FUNCTION_BLOCK ConveyorManualISub (* Conveyor Manual Interface subscribe *)
  (* Standard: 61499-2 *)
  (* Version 0.2, 2003-12-05, JHC, Rockwell Automation, Renamed from NEWCOMPFB. *)
  (* Version 0.1, 2002-01-08, JHC, Rockwell Automation, Added DLY FB as example. *)
  (* Version 0.0, 2000-05-27, JHC, Rockwell Automation *)
  (* Compiler header: package fb.rt.dasdA1.A2.Conveyor; *)
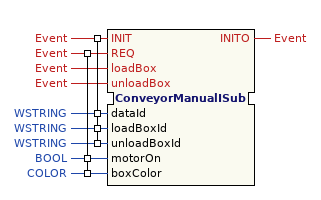
  EVENT_INPUT
    INIT WITH dataId, loadBoxId, unloadBoxId; (* Initialization Request *)
    REQ WITH motorOn, boxColor;
    loadBox;
    unloadBox;
  END_EVENT
  EVENT_OUTPUT
    INITO; (* Initialization Confirm *)
  END_EVENT
  VAR_INPUT
    dataId : WSTRING;
    loadBoxId : WSTRING;
    unloadBoxId : WSTRING;
    motorOn : BOOL;
    boxColor : COLOR;
  END_VAR
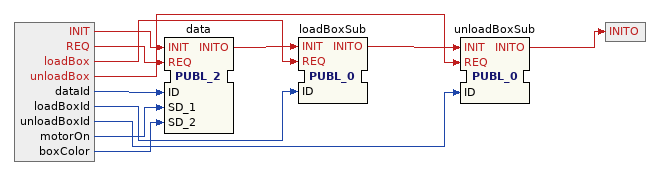
  FBS
    data : PUBL_2;
    loadBoxSub : PUBL_0;
    unloadBoxSub : PUBL_0;
  END_FBS
  EVENT_CONNECTIONS
    INIT TO data.INIT;
    REQ TO data.REQ;
    data.INITO TO loadBoxSub.INIT;
    loadBox TO loadBoxSub.REQ;
    loadBoxSub.INITO TO unloadBoxSub.INIT;
    unloadBox TO unloadBoxSub.REQ;
    unloadBoxSub.INITO TO INITO;
  END_CONNECTIONS
  DATA_CONNECTIONS
    dataId TO data.ID;
    motorOn TO data.SD_1;
    boxColor TO data.SD_2;
    loadBoxId TO loadBoxSub.ID;
    unloadBoxId TO unloadBoxSub.ID;
  END_CONNECTIONS
END_FUNCTION_BLOCK
